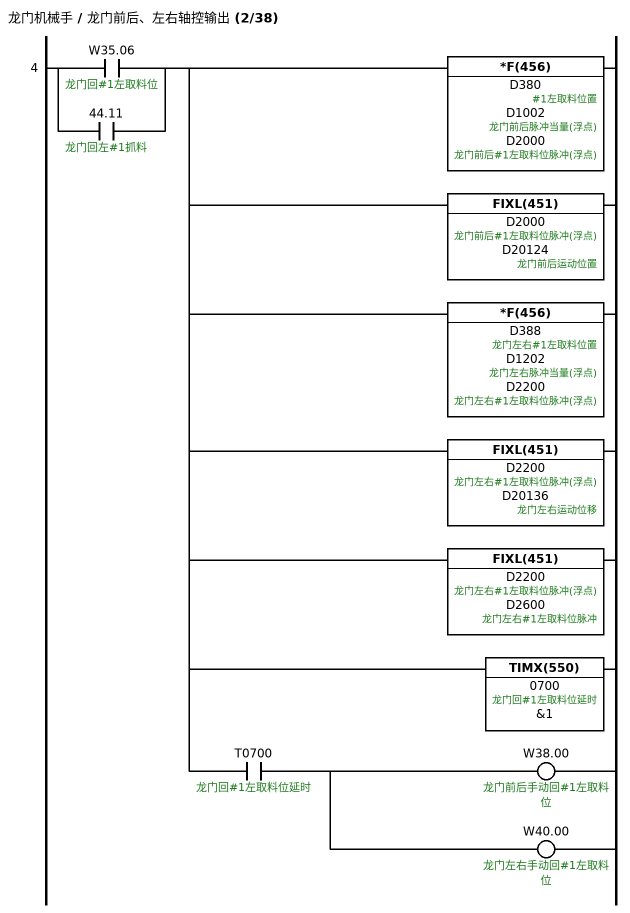
; [picture p329: 龙门机械手 / 龙门前后、左右轴控输出, rungs 4-4]
; rung 4
LD W35.06  ; 龙门回#1左取料位
OR 44.11  ; 龙门回左#1抓料
*F(456) D380 D1002 D2000  ; #1左取料位置, 龙门前后脉冲当量(浮点), 龙门前后#1左取料位脉冲(浮点)
FIXL(451) D2000 D20124  ; 龙门前后#1左取料位脉冲(浮点), 龙门前后运动位置
*F(456) D388 D1202 D2200  ; 龙门左右#1左取料位置, 龙门左右脉冲当量(浮点), 龙门左右#1左取料位脉冲(浮点)
FIXL(451) D2200 D20136  ; 龙门左右#1左取料位脉冲(浮点), 龙门左右运动位移
FIXL(451) D2200 D2600  ; 龙门左右#1左取料位脉冲(浮点), 龙门左右#1左取料位脉冲
TIMX(550) 0700 &1  ; 龙门回#1左取料位延时
AND T0700  ; 龙门回#1左取料位延时
OUT W38.00  ; 龙门前后手动回#1左取料位
OUT W40.00  ; 龙门左右手动回#1左取料位

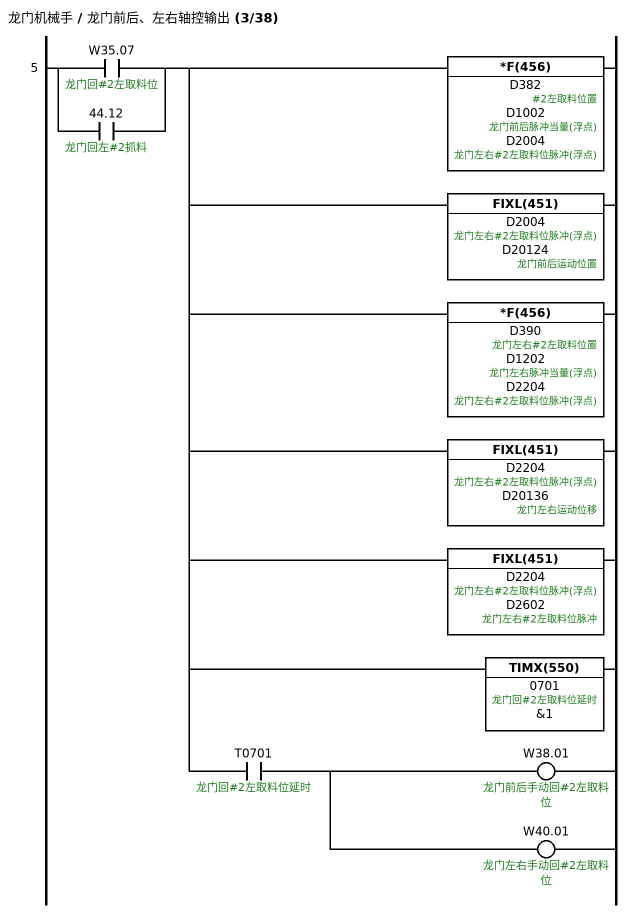
; rung 5
LD W35.07  ; 龙门回#2左取料位
OR 44.12  ; 龙门回左#2抓料
*F(456) D382 D1002 D2004  ; #2左取料位置, 龙门前后脉冲当量(浮点), 龙门左右#2左取料位脉冲(浮点)
FIXL(451) D2004 D20124  ; 龙门左右#2左取料位脉冲(浮点), 龙门前后运动位置
*F(456) D390 D1202 D2204  ; 龙门左右#2左取料位置, 龙门左右脉冲当量(浮点), 龙门左右#2左取料位脉冲(浮点)
FIXL(451) D2204 D20136  ; 龙门左右#2左取料位脉冲(浮点), 龙门左右运动位移
FIXL(451) D2204 D2602  ; 龙门左右#2左取料位脉冲(浮点), 龙门左右#2左取料位脉冲
TIMX(550) 0701 &1  ; 龙门回#2左取料位延时
AND T0701  ; 龙门回#2左取料位延时
OUT W38.01  ; 龙门前后手动回#2左取料位
OUT W40.01  ; 龙门左右手动回#2左取料位

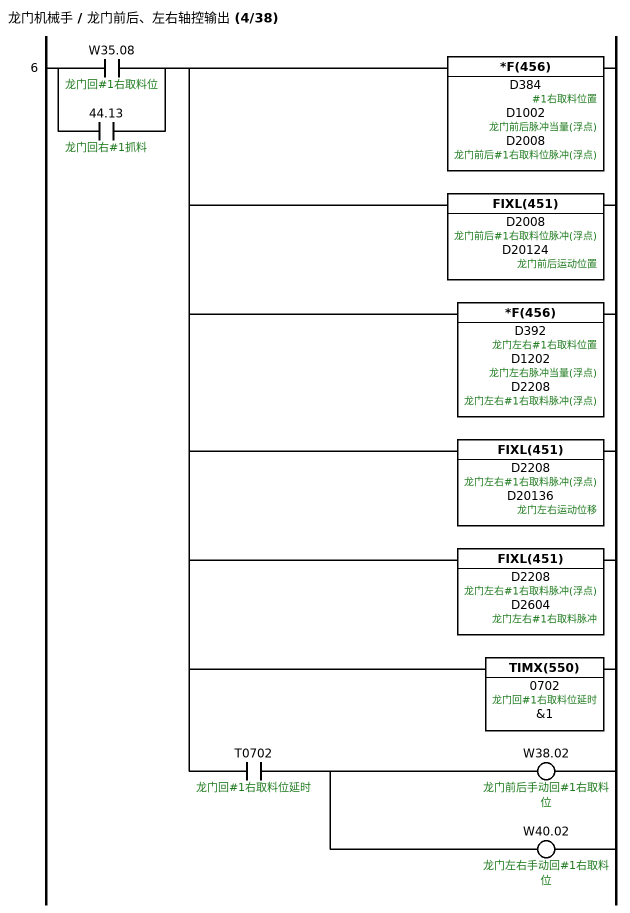
; rung 6
LD W35.08  ; 龙门回#1右取料位
OR 44.13  ; 龙门回右#1抓料
*F(456) D384 D1002 D2008  ; #1右取料位置, 龙门前后脉冲当量(浮点), 龙门前后#1右取料位脉冲(浮点)
FIXL(451) D2008 D20124  ; 龙门前后#1右取料位脉冲(浮点), 龙门前后运动位置
*F(456) D392 D1202 D2208  ; 龙门左右#1右取料位置, 龙门左右脉冲当量(浮点), 龙门左右#1右取料脉冲(浮点)
FIXL(451) D2208 D20136  ; 龙门左右#1右取料脉冲(浮点), 龙门左右运动位移
FIXL(451) D2208 D2604  ; 龙门左右#1右取料脉冲(浮点), 龙门左右#1右取料脉冲
TIMX(550) 0702 &1  ; 龙门回#1右取料位延时
AND T0702  ; 龙门回#1右取料位延时
OUT W38.02  ; 龙门前后手动回#1右取料位
OUT W40.02  ; 龙门左右手动回#1右取料位

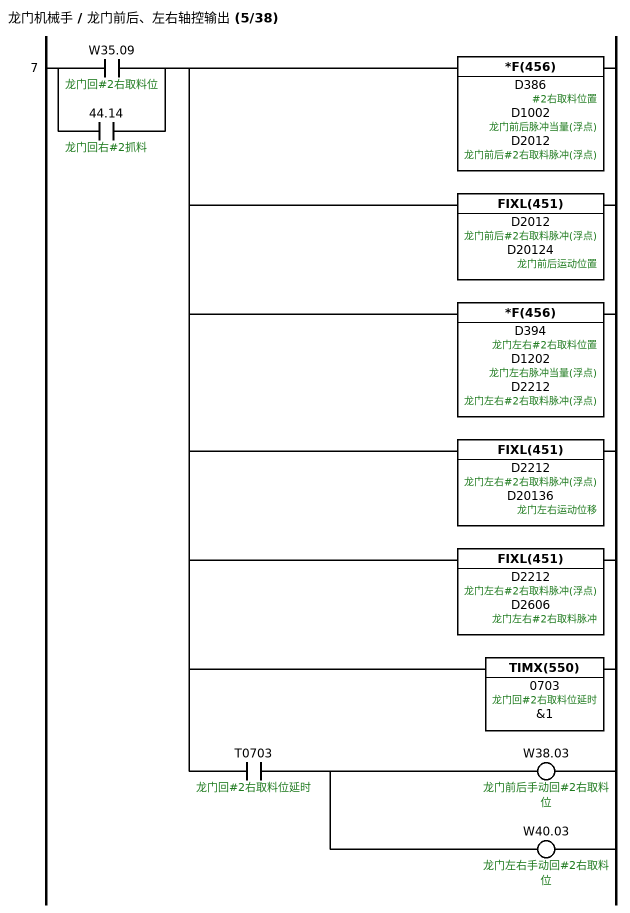
; rung 7
LD W35.09  ; 龙门回#2右取料位
OR 44.14  ; 龙门回右#2抓料
*F(456) D386 D1002 D2012  ; #2右取料位置, 龙门前后脉冲当量(浮点), 龙门前后#2右取料脉冲(浮点)
FIXL(451) D2012 D20124  ; 龙门前后#2右取料脉冲(浮点), 龙门前后运动位置
*F(456) D394 D1202 D2212  ; 龙门左右#2右取料位置, 龙门左右脉冲当量(浮点), 龙门左右#2右取料脉冲(浮点)
FIXL(451) D2212 D20136  ; 龙门左右#2右取料脉冲(浮点), 龙门左右运动位移
FIXL(451) D2212 D2606  ; 龙门左右#2右取料脉冲(浮点), 龙门左右#2右取料脉冲
TIMX(550) 0703 &1  ; 龙门回#2右取料位延时
AND T0703  ; 龙门回#2右取料位延时
OUT W38.03  ; 龙门前后手动回#2右取料位
OUT W40.03  ; 龙门左右手动回#2右取料位

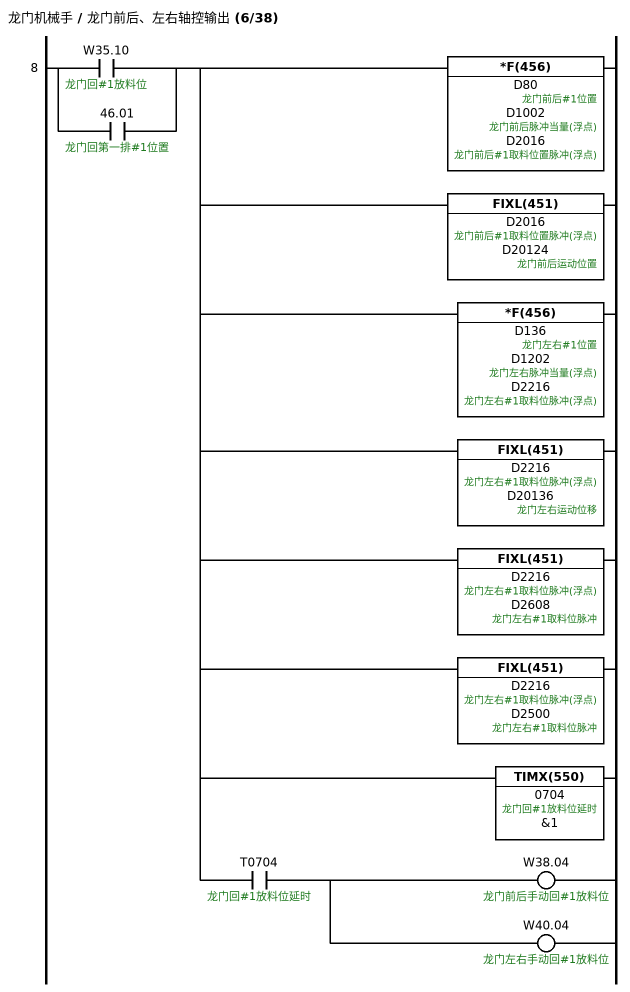
; rung 8
LD W35.10  ; 龙门回#1放料位
OR 46.01  ; 龙门回第一排#1位置
*F(456) D80 D1002 D2016  ; 龙门前后#1位置, 龙门前后脉冲当量(浮点), 龙门前后#1取料位置脉冲(浮点)
FIXL(451) D2016 D20124  ; 龙门前后#1取料位置脉冲(浮点), 龙门前后运动位置
*F(456) D136 D1202 D2216  ; 龙门左右#1位置, 龙门左右脉冲当量(浮点), 龙门左右#1取料位脉冲(浮点)
FIXL(451) D2216 D20136  ; 龙门左右#1取料位脉冲(浮点), 龙门左右运动位移
FIXL(451) D2216 D2608  ; 龙门左右#1取料位脉冲(浮点), 龙门左右#1取料位脉冲
FIXL(451) D2216 D2500  ; 龙门左右#1取料位脉冲(浮点), 龙门左右#1取料位脉冲
TIMX(550) 0704 &1  ; 龙门回#1放料位延时
AND T0704  ; 龙门回#1放料位延时
OUT W38.04  ; 龙门前后手动回#1放料位
OUT W40.04  ; 龙门左右手动回#1放料位

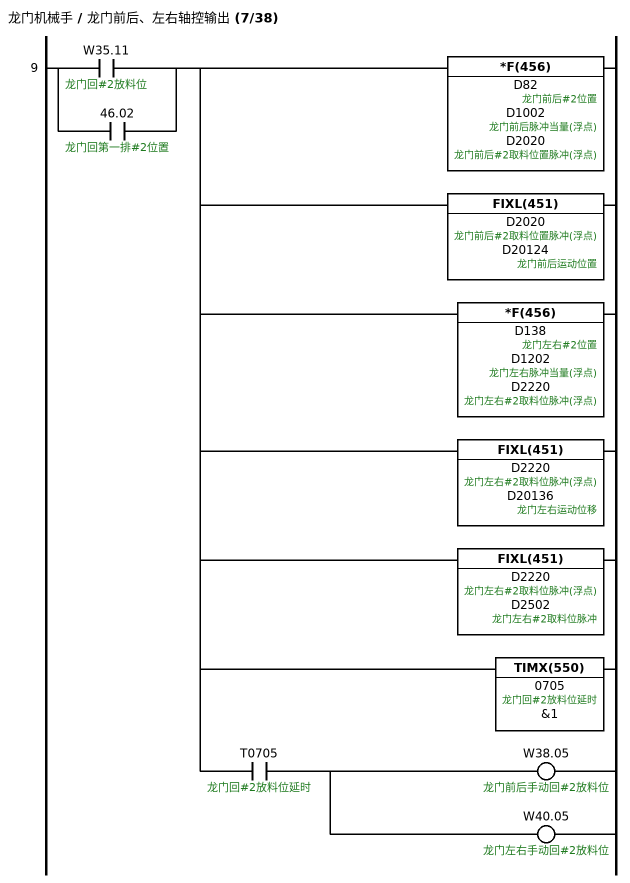
; rung 9
LD W35.11  ; 龙门回#2放料位
OR 46.02  ; 龙门回第一排#2位置
*F(456) D82 D1002 D2020  ; 龙门前后#2位置, 龙门前后脉冲当量(浮点), 龙门前后#2取料位置脉冲(浮点)
FIXL(451) D2020 D20124  ; 龙门前后#2取料位置脉冲(浮点), 龙门前后运动位置
*F(456) D138 D1202 D2220  ; 龙门左右#2位置, 龙门左右脉冲当量(浮点), 龙门左右#2取料位脉冲(浮点)
FIXL(451) D2220 D20136  ; 龙门左右#2取料位脉冲(浮点), 龙门左右运动位移
FIXL(451) D2220 D2502  ; 龙门左右#2取料位脉冲(浮点), 龙门左右#2取料位脉冲
TIMX(550) 0705 &1  ; 龙门回#2放料位延时
AND T0705  ; 龙门回#2放料位延时
OUT W38.05  ; 龙门前后手动回#2放料位
OUT W40.05  ; 龙门左右手动回#2放料位

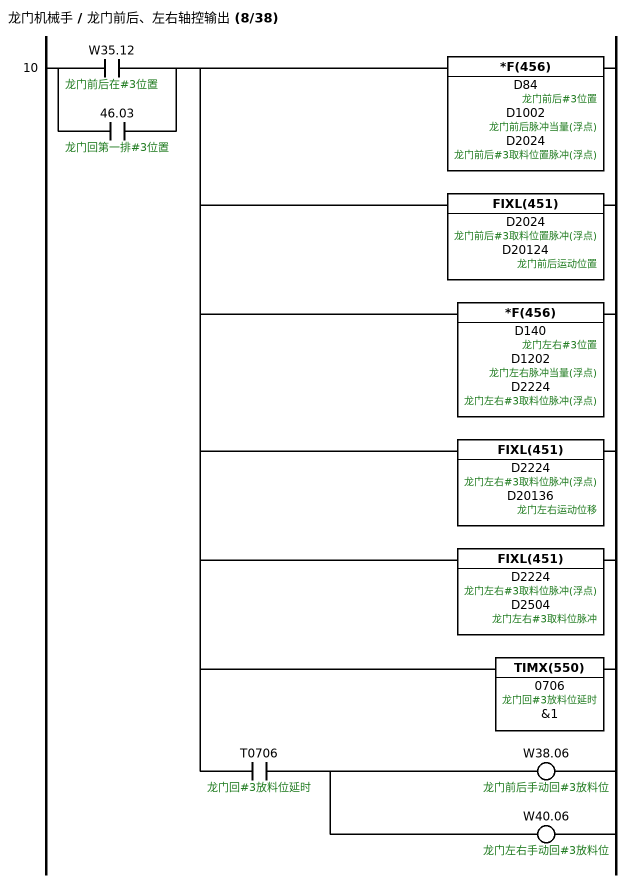
; rung 10
LD W35.12  ; 龙门前后在#3位置
OR 46.03  ; 龙门回第一排#3位置
*F(456) D84 D1002 D2024  ; 龙门前后#3位置, 龙门前后脉冲当量(浮点), 龙门前后#3取料位置脉冲(浮点)
FIXL(451) D2024 D20124  ; 龙门前后#3取料位置脉冲(浮点), 龙门前后运动位置
*F(456) D140 D1202 D2224  ; 龙门左右#3位置, 龙门左右脉冲当量(浮点), 龙门左右#3取料位脉冲(浮点)
FIXL(451) D2224 D20136  ; 龙门左右#3取料位脉冲(浮点), 龙门左右运动位移
FIXL(451) D2224 D2504  ; 龙门左右#3取料位脉冲(浮点), 龙门左右#3取料位脉冲
TIMX(550) 0706 &1  ; 龙门回#3放料位延时
AND T0706  ; 龙门回#3放料位延时
OUT W38.06  ; 龙门前后手动回#3放料位
OUT W40.06  ; 龙门左右手动回#3放料位

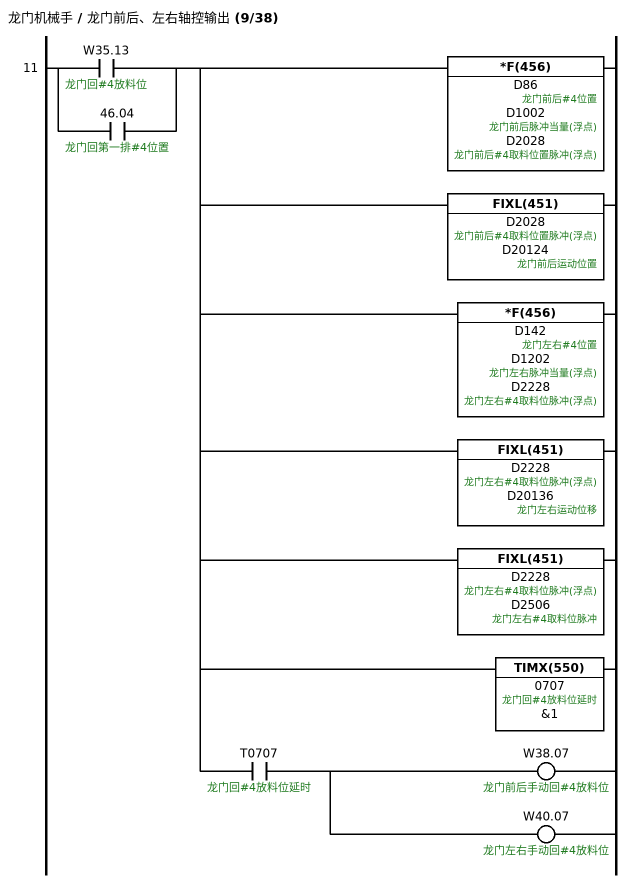
; rung 11
LD W35.13  ; 龙门回#4放料位
OR 46.04  ; 龙门回第一排#4位置
*F(456) D86 D1002 D2028  ; 龙门前后#4位置, 龙门前后脉冲当量(浮点), 龙门前后#4取料位置脉冲(浮点)
FIXL(451) D2028 D20124  ; 龙门前后#4取料位置脉冲(浮点), 龙门前后运动位置
*F(456) D142 D1202 D2228  ; 龙门左右#4位置, 龙门左右脉冲当量(浮点), 龙门左右#4取料位脉冲(浮点)
FIXL(451) D2228 D20136  ; 龙门左右#4取料位脉冲(浮点), 龙门左右运动位移
FIXL(451) D2228 D2506  ; 龙门左右#4取料位脉冲(浮点), 龙门左右#4取料位脉冲
TIMX(550) 0707 &1  ; 龙门回#4放料位延时
AND T0707  ; 龙门回#4放料位延时
OUT W38.07  ; 龙门前后手动回#4放料位
OUT W40.07  ; 龙门左右手动回#4放料位

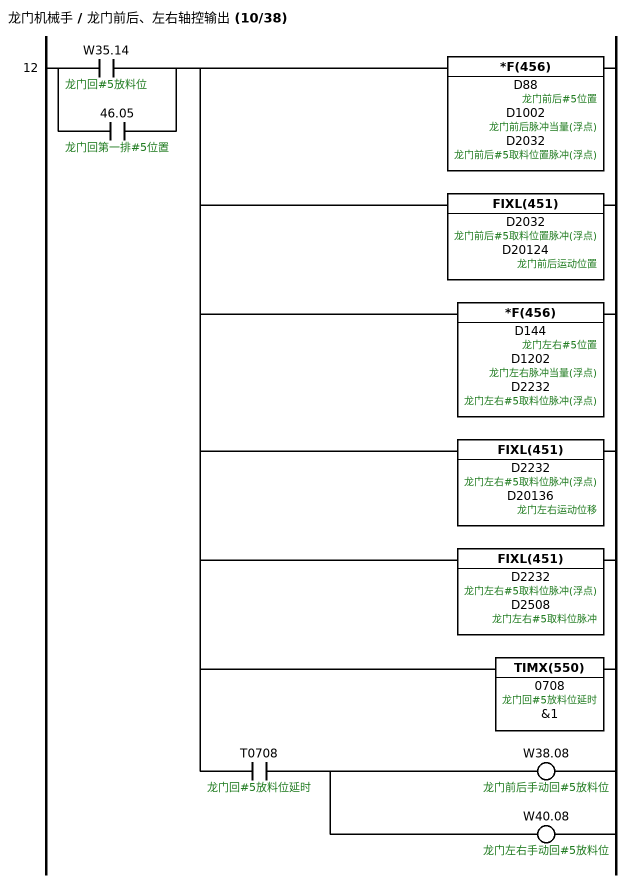
; rung 12
LD W35.14  ; 龙门回#5放料位
OR 46.05  ; 龙门回第一排#5位置
*F(456) D88 D1002 D2032  ; 龙门前后#5位置, 龙门前后脉冲当量(浮点), 龙门前后#5取料位置脉冲(浮点)
FIXL(451) D2032 D20124  ; 龙门前后#5取料位置脉冲(浮点), 龙门前后运动位置
*F(456) D144 D1202 D2232  ; 龙门左右#5位置, 龙门左右脉冲当量(浮点), 龙门左右#5取料位脉冲(浮点)
FIXL(451) D2232 D20136  ; 龙门左右#5取料位脉冲(浮点), 龙门左右运动位移
FIXL(451) D2232 D2508  ; 龙门左右#5取料位脉冲(浮点), 龙门左右#5取料位脉冲
TIMX(550) 0708 &1  ; 龙门回#5放料位延时
AND T0708  ; 龙门回#5放料位延时
OUT W38.08  ; 龙门前后手动回#5放料位
OUT W40.08  ; 龙门左右手动回#5放料位

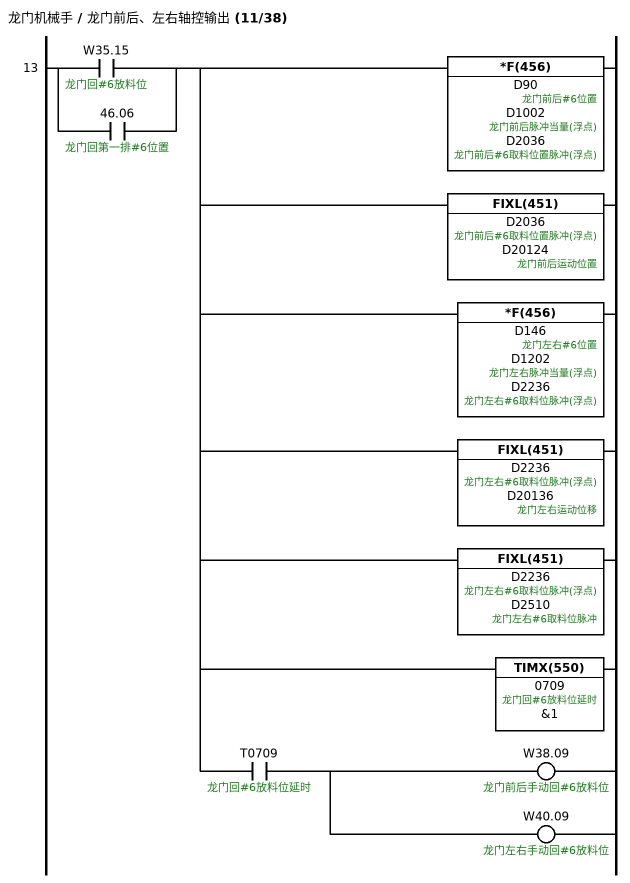
; rung 13
LD W35.15  ; 龙门回#6放料位
OR 46.06  ; 龙门回第一排#6位置
*F(456) D90 D1002 D2036  ; 龙门前后#6位置, 龙门前后脉冲当量(浮点), 龙门前后#6取料位置脉冲(浮点)
FIXL(451) D2036 D20124  ; 龙门前后#6取料位置脉冲(浮点), 龙门前后运动位置
*F(456) D146 D1202 D2236  ; 龙门左右#6位置, 龙门左右脉冲当量(浮点), 龙门左右#6取料位脉冲(浮点)
FIXL(451) D2236 D20136  ; 龙门左右#6取料位脉冲(浮点), 龙门左右运动位移
FIXL(451) D2236 D2510  ; 龙门左右#6取料位脉冲(浮点), 龙门左右#6取料位脉冲
TIMX(550) 0709 &1  ; 龙门回#6放料位延时
AND T0709  ; 龙门回#6放料位延时
OUT W38.09  ; 龙门前后手动回#6放料位
OUT W40.09  ; 龙门左右手动回#6放料位

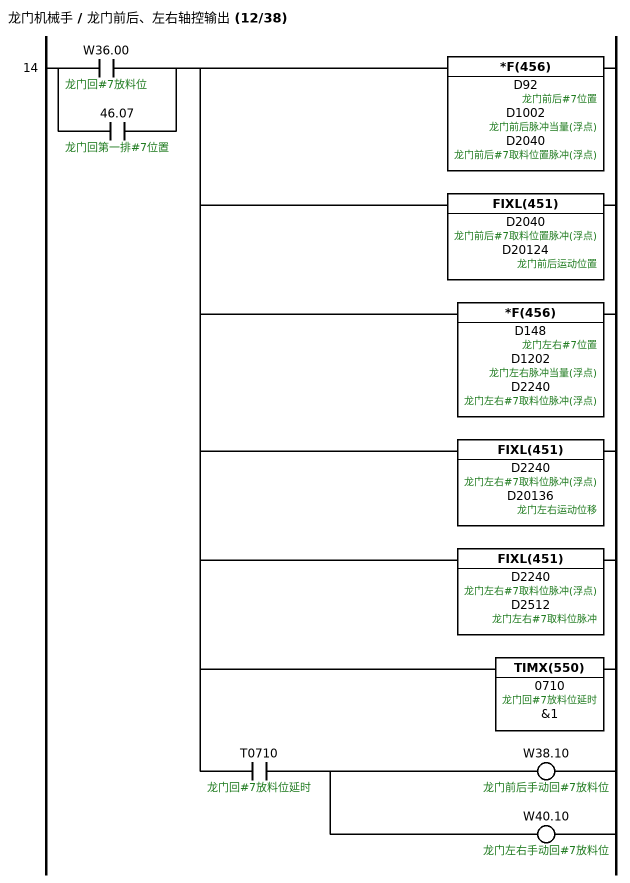
; rung 14
LD W36.00  ; 龙门回#7放料位
OR 46.07  ; 龙门回第一排#7位置
*F(456) D92 D1002 D2040  ; 龙门前后#7位置, 龙门前后脉冲当量(浮点), 龙门前后#7取料位置脉冲(浮点)
FIXL(451) D2040 D20124  ; 龙门前后#7取料位置脉冲(浮点), 龙门前后运动位置
*F(456) D148 D1202 D2240  ; 龙门左右#7位置, 龙门左右脉冲当量(浮点), 龙门左右#7取料位脉冲(浮点)
FIXL(451) D2240 D20136  ; 龙门左右#7取料位脉冲(浮点), 龙门左右运动位移
FIXL(451) D2240 D2512  ; 龙门左右#7取料位脉冲(浮点), 龙门左右#7取料位脉冲
TIMX(550) 0710 &1  ; 龙门回#7放料位延时
AND T0710  ; 龙门回#7放料位延时
OUT W38.10  ; 龙门前后手动回#7放料位
OUT W40.10  ; 龙门左右手动回#7放料位

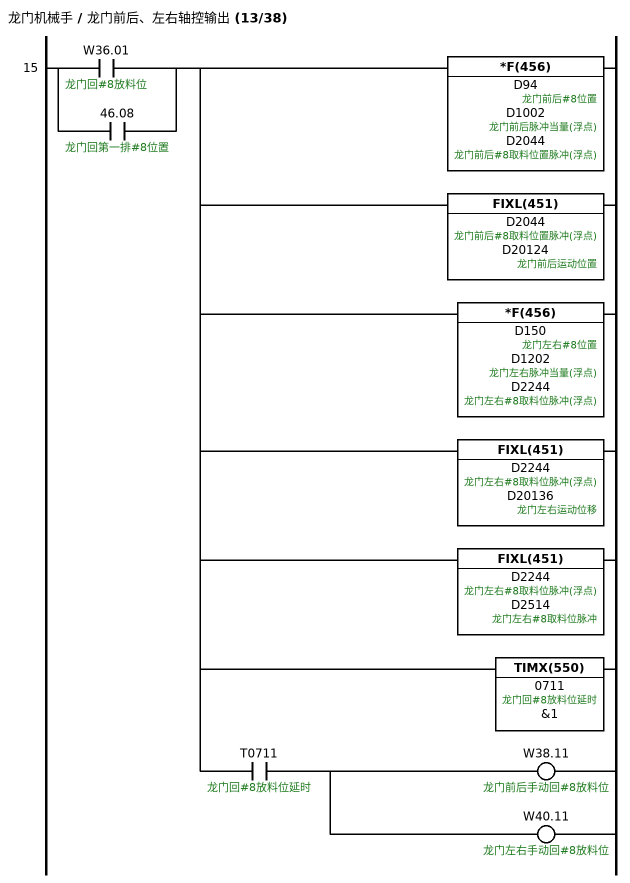
; rung 15
LD W36.01  ; 龙门回#8放料位
OR 46.08  ; 龙门回第一排#8位置
*F(456) D94 D1002 D2044  ; 龙门前后#8位置, 龙门前后脉冲当量(浮点), 龙门前后#8取料位置脉冲(浮点)
FIXL(451) D2044 D20124  ; 龙门前后#8取料位置脉冲(浮点), 龙门前后运动位置
*F(456) D150 D1202 D2244  ; 龙门左右#8位置, 龙门左右脉冲当量(浮点), 龙门左右#8取料位脉冲(浮点)
FIXL(451) D2244 D20136  ; 龙门左右#8取料位脉冲(浮点), 龙门左右运动位移
FIXL(451) D2244 D2514  ; 龙门左右#8取料位脉冲(浮点), 龙门左右#8取料位脉冲
TIMX(550) 0711 &1  ; 龙门回#8放料位延时
AND T0711  ; 龙门回#8放料位延时
OUT W38.11  ; 龙门前后手动回#8放料位
OUT W40.11  ; 龙门左右手动回#8放料位

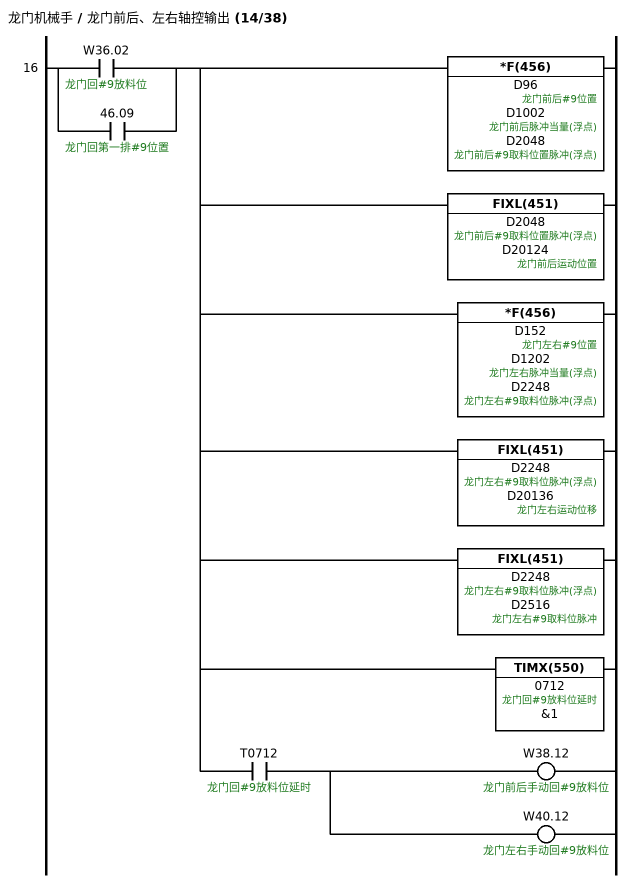
; rung 16
LD W36.02  ; 龙门回#9放料位
OR 46.09  ; 龙门回第一排#9位置
*F(456) D96 D1002 D2048  ; 龙门前后#9位置, 龙门前后脉冲当量(浮点), 龙门前后#9取料位置脉冲(浮点)
FIXL(451) D2048 D20124  ; 龙门前后#9取料位置脉冲(浮点), 龙门前后运动位置
*F(456) D152 D1202 D2248  ; 龙门左右#9位置, 龙门左右脉冲当量(浮点), 龙门左右#9取料位脉冲(浮点)
FIXL(451) D2248 D20136  ; 龙门左右#9取料位脉冲(浮点), 龙门左右运动位移
FIXL(451) D2248 D2516  ; 龙门左右#9取料位脉冲(浮点), 龙门左右#9取料位脉冲
TIMX(550) 0712 &1  ; 龙门回#9放料位延时
AND T0712  ; 龙门回#9放料位延时
OUT W38.12  ; 龙门前后手动回#9放料位
OUT W40.12  ; 龙门左右手动回#9放料位

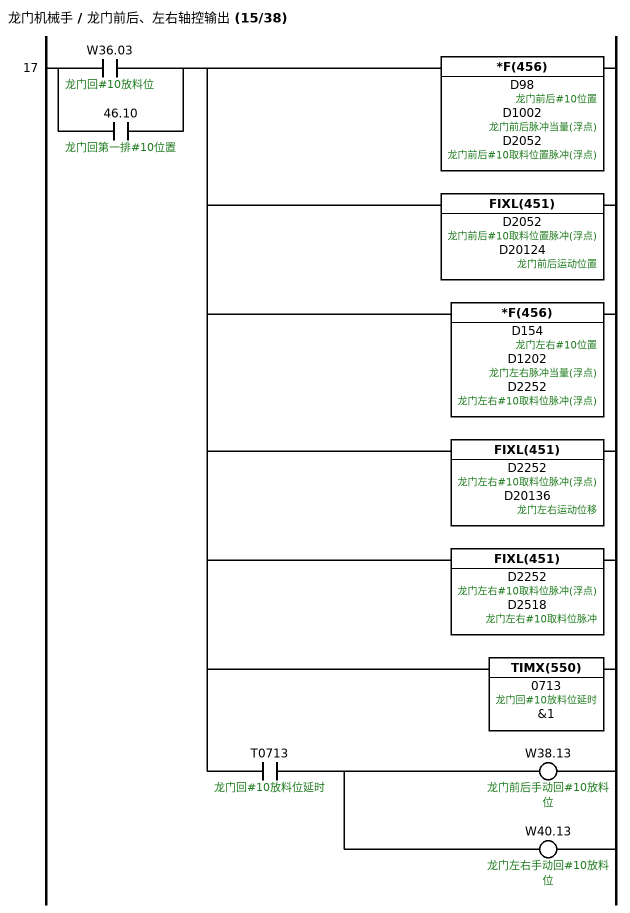
; rung 17
LD W36.03  ; 龙门回#10放料位
OR 46.10  ; 龙门回第一排#10位置
*F(456) D98 D1002 D2052  ; 龙门前后#10位置, 龙门前后脉冲当量(浮点), 龙门前后#10取料位置脉冲(浮点)
FIXL(451) D2052 D20124  ; 龙门前后#10取料位置脉冲(浮点), 龙门前后运动位置
*F(456) D154 D1202 D2252  ; 龙门左右#10位置, 龙门左右脉冲当量(浮点), 龙门左右#10取料位脉冲(浮点)
FIXL(451) D2252 D20136  ; 龙门左右#10取料位脉冲(浮点), 龙门左右运动位移
FIXL(451) D2252 D2518  ; 龙门左右#10取料位脉冲(浮点), 龙门左右#10取料位脉冲
TIMX(550) 0713 &1  ; 龙门回#10放料位延时
AND T0713  ; 龙门回#10放料位延时
OUT W38.13  ; 龙门前后手动回#10放料位
OUT W40.13  ; 龙门左右手动回#10放料位

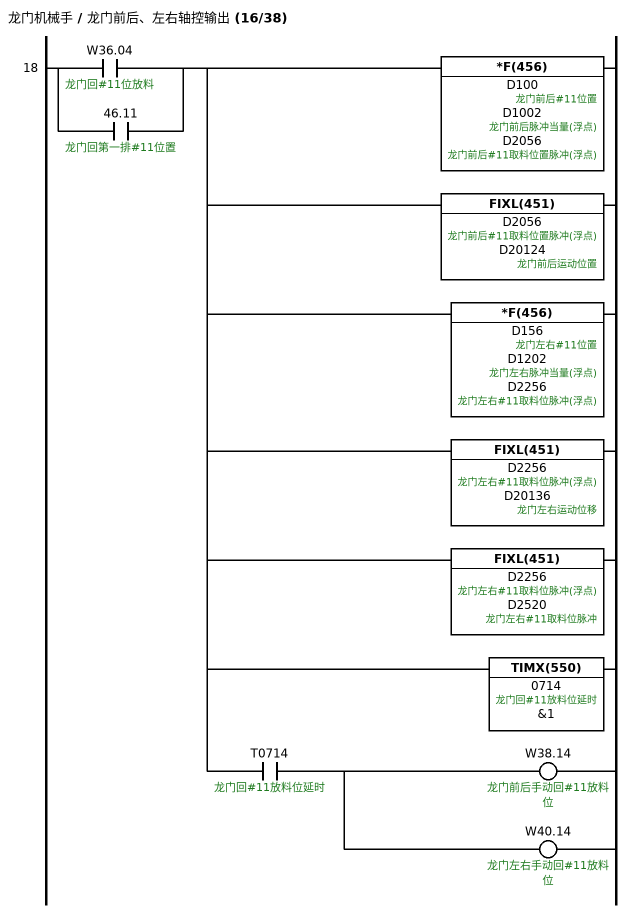
; rung 18
LD W36.04  ; 龙门回#11位放料
OR 46.11  ; 龙门回第一排#11位置
*F(456) D100 D1002 D2056  ; 龙门前后#11位置, 龙门前后脉冲当量(浮点), 龙门前后#11取料位置脉冲(浮点)
FIXL(451) D2056 D20124  ; 龙门前后#11取料位置脉冲(浮点), 龙门前后运动位置
*F(456) D156 D1202 D2256  ; 龙门左右#11位置, 龙门左右脉冲当量(浮点), 龙门左右#11取料位脉冲(浮点)
FIXL(451) D2256 D20136  ; 龙门左右#11取料位脉冲(浮点), 龙门左右运动位移
FIXL(451) D2256 D2520  ; 龙门左右#11取料位脉冲(浮点), 龙门左右#11取料位脉冲
TIMX(550) 0714 &1  ; 龙门回#11放料位延时
AND T0714  ; 龙门回#11放料位延时
OUT W38.14  ; 龙门前后手动回#11放料位
OUT W40.14  ; 龙门左右手动回#11放料位

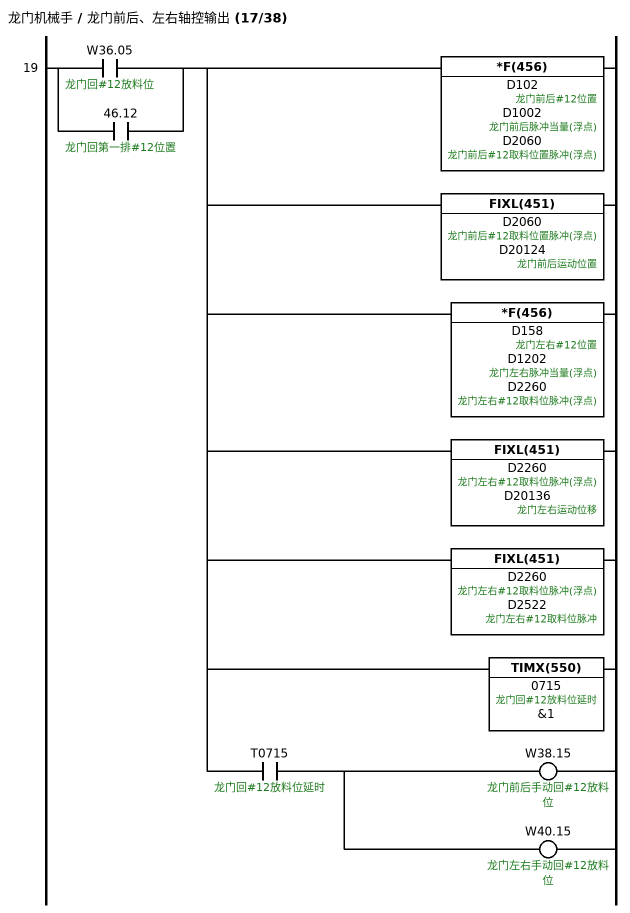
; rung 19
LD W36.05  ; 龙门回#12放料位
OR 46.12  ; 龙门回第一排#12位置
*F(456) D102 D1002 D2060  ; 龙门前后#12位置, 龙门前后脉冲当量(浮点), 龙门前后#12取料位置脉冲(浮点)
FIXL(451) D2060 D20124  ; 龙门前后#12取料位置脉冲(浮点), 龙门前后运动位置
*F(456) D158 D1202 D2260  ; 龙门左右#12位置, 龙门左右脉冲当量(浮点), 龙门左右#12取料位脉冲(浮点)
FIXL(451) D2260 D20136  ; 龙门左右#12取料位脉冲(浮点), 龙门左右运动位移
FIXL(451) D2260 D2522  ; 龙门左右#12取料位脉冲(浮点), 龙门左右#12取料位脉冲
TIMX(550) 0715 &1  ; 龙门回#12放料位延时
AND T0715  ; 龙门回#12放料位延时
OUT W38.15  ; 龙门前后手动回#12放料位
OUT W40.15  ; 龙门左右手动回#12放料位

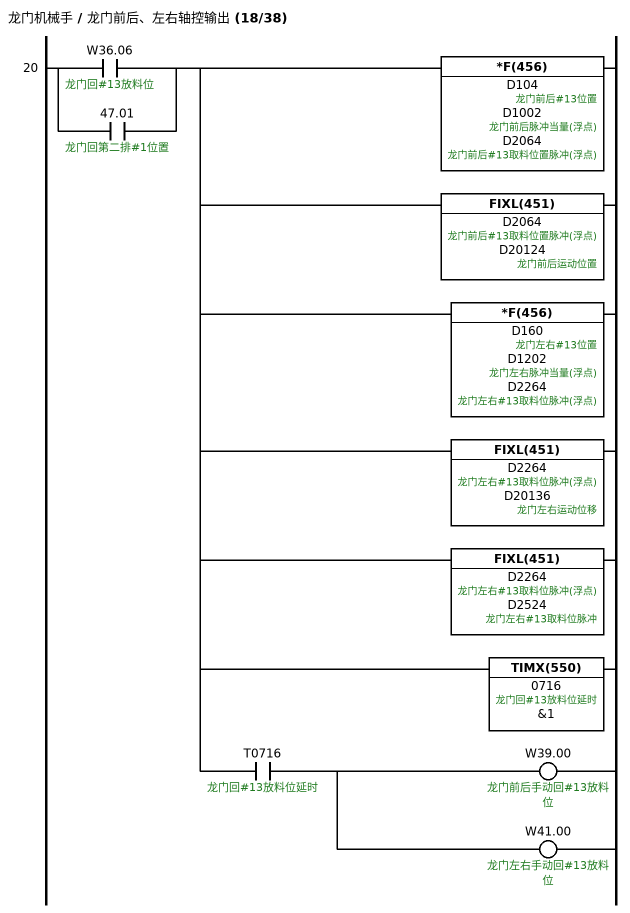
; rung 20
LD W36.06  ; 龙门回#13放料位
OR 47.01  ; 龙门回第二排#1位置
*F(456) D104 D1002 D2064  ; 龙门前后#13位置, 龙门前后脉冲当量(浮点), 龙门前后#13取料位置脉冲(浮点)
FIXL(451) D2064 D20124  ; 龙门前后#13取料位置脉冲(浮点), 龙门前后运动位置
*F(456) D160 D1202 D2264  ; 龙门左右#13位置, 龙门左右脉冲当量(浮点), 龙门左右#13取料位脉冲(浮点)
FIXL(451) D2264 D20136  ; 龙门左右#13取料位脉冲(浮点), 龙门左右运动位移
FIXL(451) D2264 D2524  ; 龙门左右#13取料位脉冲(浮点), 龙门左右#13取料位脉冲
TIMX(550) 0716 &1  ; 龙门回#13放料位延时
AND T0716  ; 龙门回#13放料位延时
OUT W39.00  ; 龙门前后手动回#13放料位
OUT W41.00  ; 龙门左右手动回#13放料位

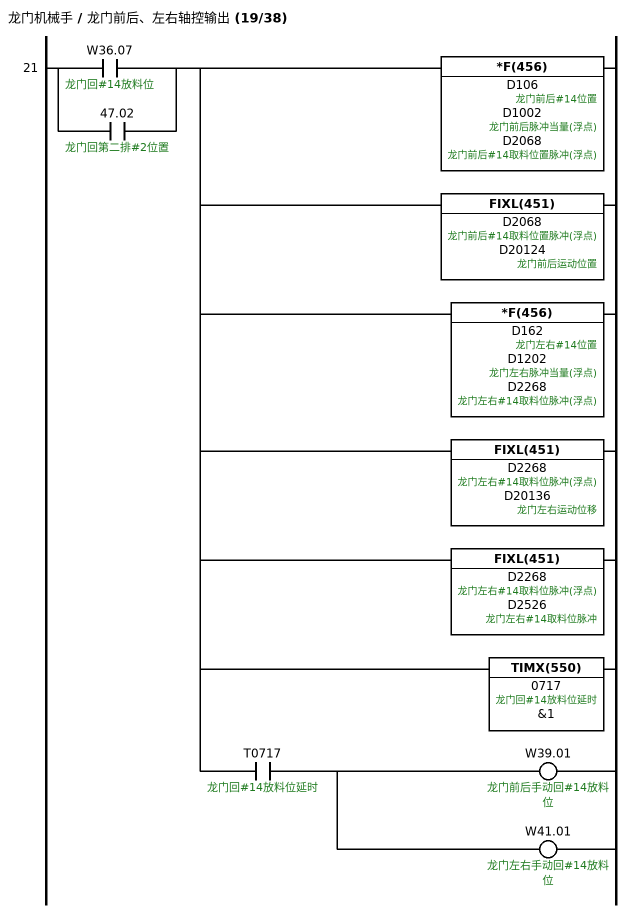
; rung 21
LD W36.07  ; 龙门回#14放料位
OR 47.02  ; 龙门回第二排#2位置
*F(456) D106 D1002 D2068  ; 龙门前后#14位置, 龙门前后脉冲当量(浮点), 龙门前后#14取料位置脉冲(浮点)
FIXL(451) D2068 D20124  ; 龙门前后#14取料位置脉冲(浮点), 龙门前后运动位置
*F(456) D162 D1202 D2268  ; 龙门左右#14位置, 龙门左右脉冲当量(浮点), 龙门左右#14取料位脉冲(浮点)
FIXL(451) D2268 D20136  ; 龙门左右#14取料位脉冲(浮点), 龙门左右运动位移
FIXL(451) D2268 D2526  ; 龙门左右#14取料位脉冲(浮点), 龙门左右#14取料位脉冲
TIMX(550) 0717 &1  ; 龙门回#14放料位延时
AND T0717  ; 龙门回#14放料位延时
OUT W39.01  ; 龙门前后手动回#14放料位
OUT W41.01  ; 龙门左右手动回#14放料位

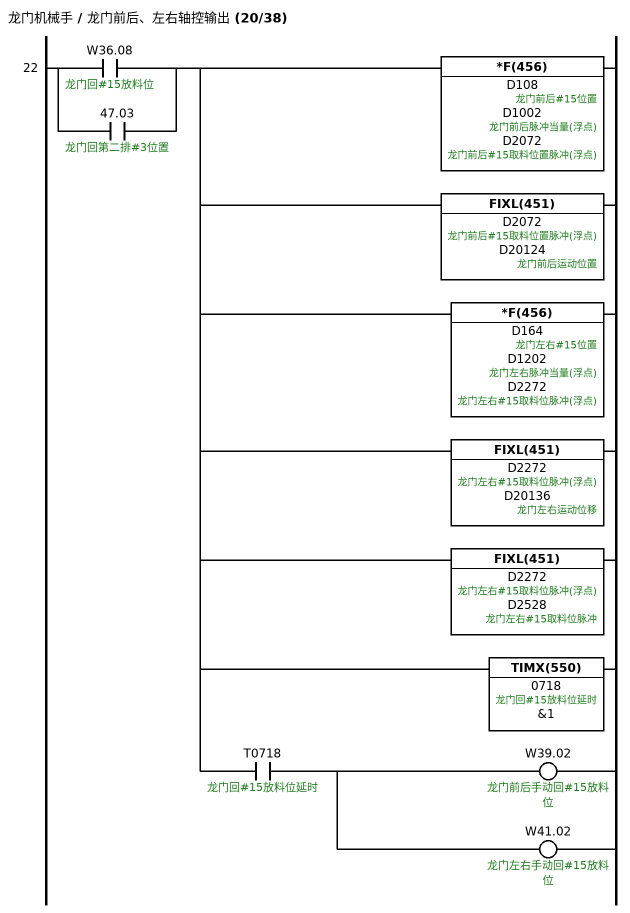
; rung 22
LD W36.08  ; 龙门回#15放料位
OR 47.03  ; 龙门回第二排#3位置
*F(456) D108 D1002 D2072  ; 龙门前后#15位置, 龙门前后脉冲当量(浮点), 龙门前后#15取料位置脉冲(浮点)
FIXL(451) D2072 D20124  ; 龙门前后#15取料位置脉冲(浮点), 龙门前后运动位置
*F(456) D164 D1202 D2272  ; 龙门左右#15位置, 龙门左右脉冲当量(浮点), 龙门左右#15取料位脉冲(浮点)
FIXL(451) D2272 D20136  ; 龙门左右#15取料位脉冲(浮点), 龙门左右运动位移
FIXL(451) D2272 D2528  ; 龙门左右#15取料位脉冲(浮点), 龙门左右#15取料位脉冲
TIMX(550) 0718 &1  ; 龙门回#15放料位延时
AND T0718  ; 龙门回#15放料位延时
OUT W39.02  ; 龙门前后手动回#15放料位
OUT W41.02  ; 龙门左右手动回#15放料位

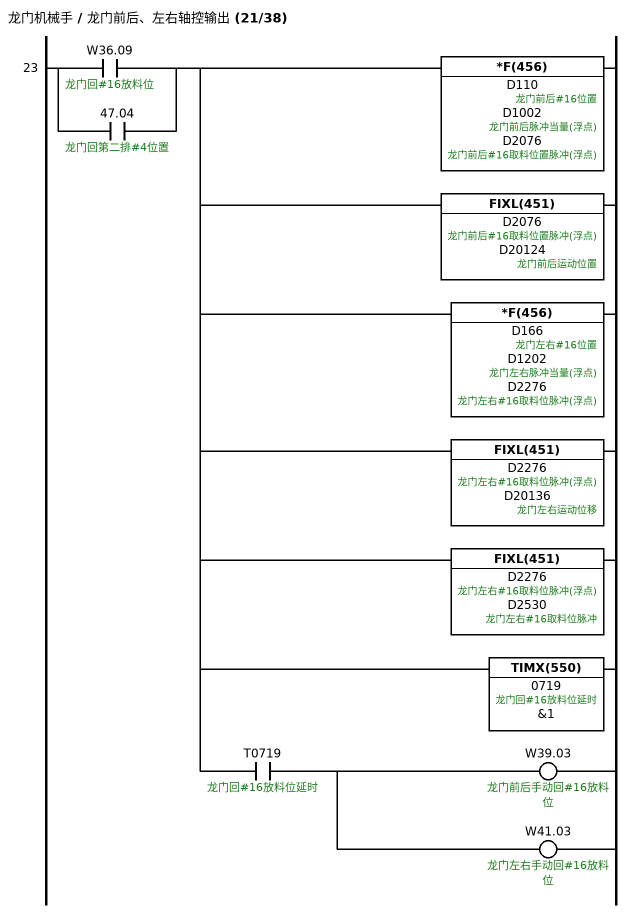
; rung 23
LD W36.09  ; 龙门回#16放料位
OR 47.04  ; 龙门回第二排#4位置
*F(456) D110 D1002 D2076  ; 龙门前后#16位置, 龙门前后脉冲当量(浮点), 龙门前后#16取料位置脉冲(浮点)
FIXL(451) D2076 D20124  ; 龙门前后#16取料位置脉冲(浮点), 龙门前后运动位置
*F(456) D166 D1202 D2276  ; 龙门左右#16位置, 龙门左右脉冲当量(浮点), 龙门左右#16取料位脉冲(浮点)
FIXL(451) D2276 D20136  ; 龙门左右#16取料位脉冲(浮点), 龙门左右运动位移
FIXL(451) D2276 D2530  ; 龙门左右#16取料位脉冲(浮点), 龙门左右#16取料位脉冲
TIMX(550) 0719 &1  ; 龙门回#16放料位延时
AND T0719  ; 龙门回#16放料位延时
OUT W39.03  ; 龙门前后手动回#16放料位
OUT W41.03  ; 龙门左右手动回#16放料位

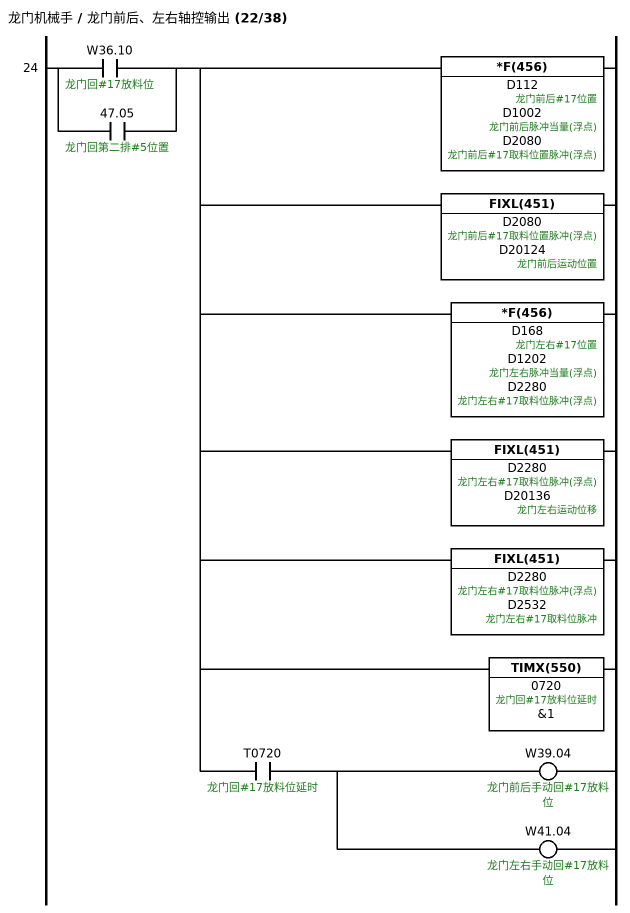
; rung 24
LD W36.10  ; 龙门回#17放料位
OR 47.05  ; 龙门回第二排#5位置
*F(456) D112 D1002 D2080  ; 龙门前后#17位置, 龙门前后脉冲当量(浮点), 龙门前后#17取料位置脉冲(浮点)
FIXL(451) D2080 D20124  ; 龙门前后#17取料位置脉冲(浮点), 龙门前后运动位置
*F(456) D168 D1202 D2280  ; 龙门左右#17位置, 龙门左右脉冲当量(浮点), 龙门左右#17取料位脉冲(浮点)
FIXL(451) D2280 D20136  ; 龙门左右#17取料位脉冲(浮点), 龙门左右运动位移
FIXL(451) D2280 D2532  ; 龙门左右#17取料位脉冲(浮点), 龙门左右#17取料位脉冲
TIMX(550) 0720 &1  ; 龙门回#17放料位延时
AND T0720  ; 龙门回#17放料位延时
OUT W39.04  ; 龙门前后手动回#17放料位
OUT W41.04  ; 龙门左右手动回#17放料位

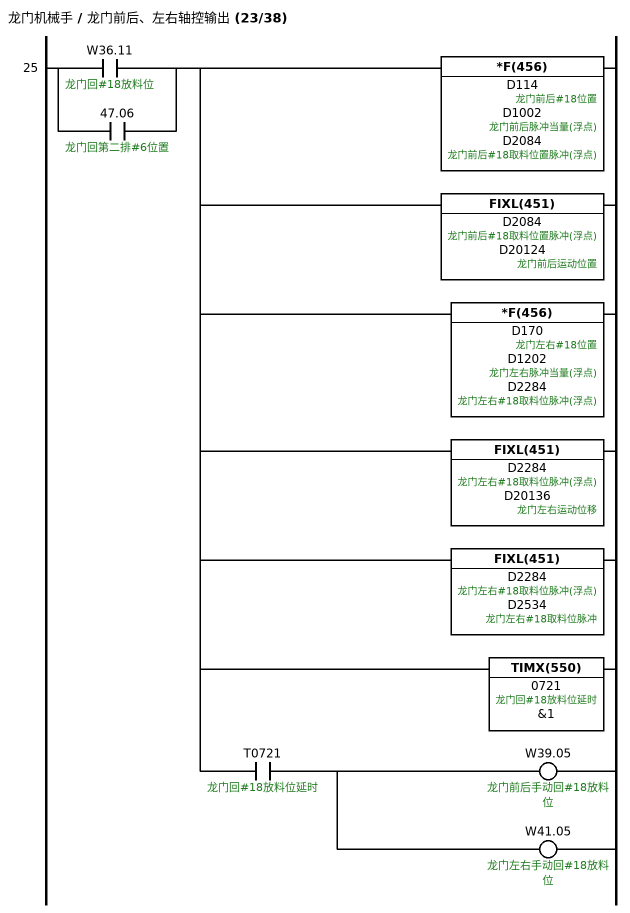
; rung 25
LD W36.11  ; 龙门回#18放料位
OR 47.06  ; 龙门回第二排#6位置
*F(456) D114 D1002 D2084  ; 龙门前后#18位置, 龙门前后脉冲当量(浮点), 龙门前后#18取料位置脉冲(浮点)
FIXL(451) D2084 D20124  ; 龙门前后#18取料位置脉冲(浮点), 龙门前后运动位置
*F(456) D170 D1202 D2284  ; 龙门左右#18位置, 龙门左右脉冲当量(浮点), 龙门左右#18取料位脉冲(浮点)
FIXL(451) D2284 D20136  ; 龙门左右#18取料位脉冲(浮点), 龙门左右运动位移
FIXL(451) D2284 D2534  ; 龙门左右#18取料位脉冲(浮点), 龙门左右#18取料位脉冲
TIMX(550) 0721 &1  ; 龙门回#18放料位延时
AND T0721  ; 龙门回#18放料位延时
OUT W39.05  ; 龙门前后手动回#18放料位
OUT W41.05  ; 龙门左右手动回#18放料位

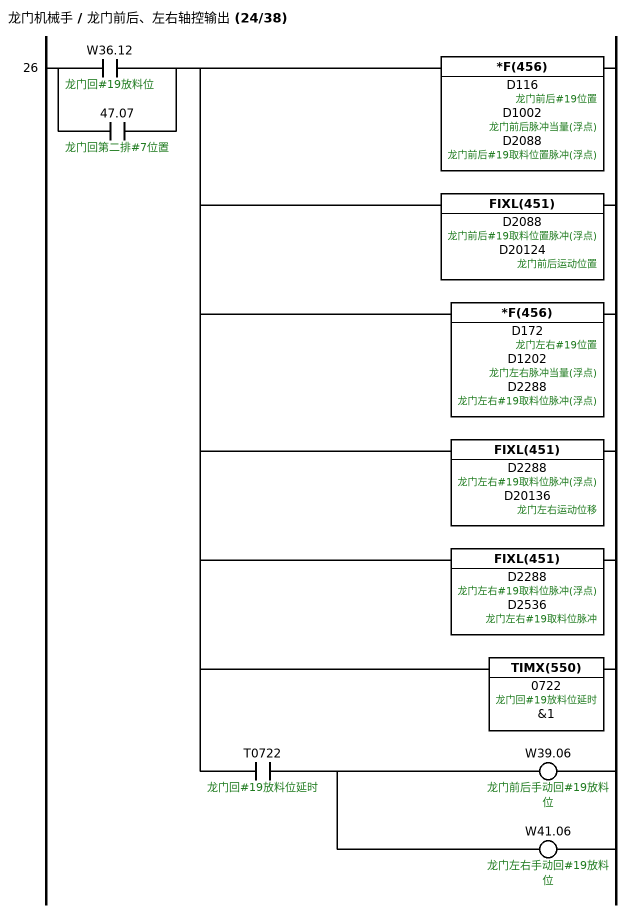
; rung 26
LD W36.12  ; 龙门回#19放料位
OR 47.07  ; 龙门回第二排#7位置
*F(456) D116 D1002 D2088  ; 龙门前后#19位置, 龙门前后脉冲当量(浮点), 龙门前后#19取料位置脉冲(浮点)
FIXL(451) D2088 D20124  ; 龙门前后#19取料位置脉冲(浮点), 龙门前后运动位置
*F(456) D172 D1202 D2288  ; 龙门左右#19位置, 龙门左右脉冲当量(浮点), 龙门左右#19取料位脉冲(浮点)
FIXL(451) D2288 D20136  ; 龙门左右#19取料位脉冲(浮点), 龙门左右运动位移
FIXL(451) D2288 D2536  ; 龙门左右#19取料位脉冲(浮点), 龙门左右#19取料位脉冲
TIMX(550) 0722 &1  ; 龙门回#19放料位延时
AND T0722  ; 龙门回#19放料位延时
OUT W39.06  ; 龙门前后手动回#19放料位
OUT W41.06  ; 龙门左右手动回#19放料位

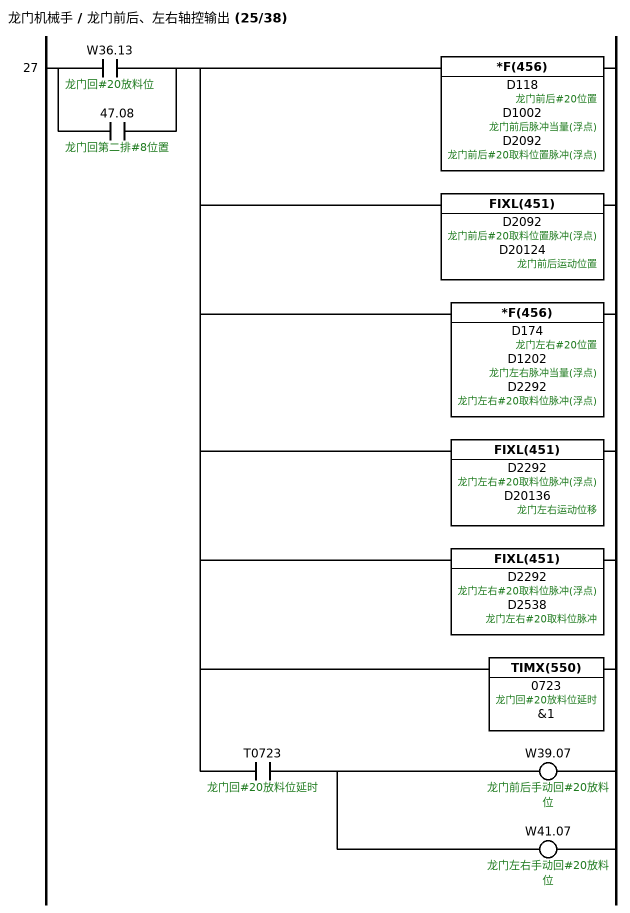
; rung 27
LD W36.13  ; 龙门回#20放料位
OR 47.08  ; 龙门回第二排#8位置
*F(456) D118 D1002 D2092  ; 龙门前后#20位置, 龙门前后脉冲当量(浮点), 龙门前后#20取料位置脉冲(浮点)
FIXL(451) D2092 D20124  ; 龙门前后#20取料位置脉冲(浮点), 龙门前后运动位置
*F(456) D174 D1202 D2292  ; 龙门左右#20位置, 龙门左右脉冲当量(浮点), 龙门左右#20取料位脉冲(浮点)
FIXL(451) D2292 D20136  ; 龙门左右#20取料位脉冲(浮点), 龙门左右运动位移
FIXL(451) D2292 D2538  ; 龙门左右#20取料位脉冲(浮点), 龙门左右#20取料位脉冲
TIMX(550) 0723 &1  ; 龙门回#20放料位延时
AND T0723  ; 龙门回#20放料位延时
OUT W39.07  ; 龙门前后手动回#20放料位
OUT W41.07  ; 龙门左右手动回#20放料位

